FUNCTION_BLOCK FB_NOTT_CO2_TRANS_STAGES
VAR_INPUT
END_VAR
VAR_OUTPUT
END_VAR
VAR
	NCP1:		FB_NOTT_MOTOR;
	NCP2:		FB_NOTT_MOTOR;
	NCP3:		FB_NOTT_MOTOR;
	NCP4:		FB_NOTT_MOTOR;
	
	
	ptrNCPs:	ARRAY [1..4] OF POINTER TO FB_NOTT_MOTOR;
	// GUI stuff
	guiNCPsIndex:	UINT := 1;	// Index for Shutter Engineering GUI
	
	stat:		T_NOTT_STAT;
	
END_VAR



NCP1(
	in_bSafe:=, 
	in_bDisableIfUnsafe:=, 
	sName:= 'NCP 1', 
	nNOVRAM_DevId:= 6, 
	nNOVRAM_Offset:= 25000);
	
NCP2(
	in_bSafe:=, 
	in_bDisableIfUnsafe:=, 
	sName:= 'NCP 2', 
	nNOVRAM_DevId:= 6, 
	nNOVRAM_Offset:= 26000);
	
NCP3(
	in_bSafe:=, 
	in_bDisableIfUnsafe:=, 
	sName:= 'NCP 3', 
	nNOVRAM_DevId:= 6, 
	nNOVRAM_Offset:= 27000);
	
NCP4(
	in_bSafe:=, 
	in_bDisableIfUnsafe:=, 
	sName:= 'NCP 4', 
	nNOVRAM_DevId:= 6, 
	nNOVRAM_Offset:= 28000);

	
M_Configure();

METHOD M_Configure : BOOL
VAR_INPUT
END_VAR

ptrNCPs[1] := ADR(NCP1);
ptrNCPs[2] := ADR(NCP2);
ptrNCPs[3] := ADR(NCP3);
ptrNCPs[4] := ADR(NCP4);
END_METHOD

END_FUNCTION_BLOCK

(* stored: Version 1.1.0.1, ProductVersion 3.1.4024.14
   POU FB_NOTT_CO2_TRANS_STAGES: Id {55170b58-63a0-43a4-953c-e7d76ea2abd1}, SpecialFunc None
   Method M_Configure: Id {64a7d10e-af79-4d51-8967-cb714db219d2} *)
